// TIA Portal V18 export
DATA_BLOCK "FB10-Condition Check_1_DB"   // DB283
VERSION : 0.1
// stored: AutoNumber true, DBAccessibleFromOPCUA true, InstanceOfName FB10-Condition Check_1, InstanceOfType FB
"FB10-Condition Check_1"
   // VAR_INPUT
   //    "Time" : DInt;
   //    "Pump ON delay" : DInt;
   //    Check_Time { ExternalAccessible := 'False'; ExternalVisible := 'False'; ExternalWritable := 'False'} : DInt;
   //    Pressure_SP { ExternalAccessible := 'False'; ExternalVisible := 'False'; ExternalWritable := 'False'} : Real;
   //    Pressure_tolerance { ExternalAccessible := 'False'; ExternalVisible := 'False'; ExternalWritable := 'False'} : Real;
   //    Current_pressure { ExternalAccessible := 'False'; ExternalVisible := 'False'; ExternalWritable := 'False'} : Real;
   //    selected { ExternalAccessible := 'False'; ExternalVisible := 'False'; ExternalWritable := 'False'} : Bool;
   //    "Pressurising Tolerance" : Real;
   //    Pressurising_SP : Real;
   // END_VAR
   // VAR_OUTPUT
   //    "dispensing Time PV" : Int;
   //    "Checking Time pv" { ExternalAccessible := 'False'; ExternalVisible := 'False'; ExternalWritable := 'False'} : Int;
   //    Leaktest_ok { ExternalAccessible := 'False'; ExternalVisible := 'False'; ExternalWritable := 'False'} : Bool;
   //    Leaktest_nok { ExternalAccessible := 'False'; ExternalVisible := 'False'; ExternalWritable := 'False'} : Bool;
   //    Conditiontest_OK : Bool;
   //    Conditiontest_NOK { ExternalAccessible := 'False'; ExternalVisible := 'False'; ExternalWritable := 'False'} : Bool;
   //    "PAT @ installation" : DInt;
   //    Test_Data : "Condition_Check";
   // END_VAR
   // VAR_IN_OUT
   //    Commissioning_mode : Bool;
   //    "Start ConditonCheck" : Bool;
   //    "Stop ConditonCheck" : Bool;
   //    "ConditonCheck Running" : Bool;
   //    "ConditonCheck completed" : Bool;
   //    "ON Gear Pump" : Bool;
   //    "ON inlet" : Bool;
   //    Pressurising : Bool;
   //    run_rev : Bool;
   // END_VAR
   // VAR
   //    "dispensing time done" : Bool;
   //    "dispensing time in sec" : DInt;
   //    "timer input" : DInt;
   //    IEC_Timer_0_Instance_1 { S7_SetPoint := 'True'} : TON_TIME;
   //    IEC_Timer_0_Instance_2 { S7_SetPoint := 'True'} : TON_TIME;
   //    IEC_Timer_0_Instance_4 { S7_SetPoint := 'True'} : TON_TIME;
   //    "Press+ve" { ExternalAccessible := 'False'; ExternalVisible := 'False'; ExternalWritable := 'False'; S7_SetPoint := 'True'} : Real;
   //    "Press-ve" { ExternalAccessible := 'False'; ExternalVisible := 'False'; ExternalWritable := 'False'} : Real;
   //    IEC_Timer_0_Instance_3 { ExternalAccessible := 'False'; ExternalVisible := 'False'; ExternalWritable := 'False'; S7_SetPoint := 'True'} : TON_TIME;
   //    Checktime_ms { ExternalAccessible := 'False'; ExternalVisible := 'False'; ExternalWritable := 'False'; S7_SetPoint := 'True'} : DInt;
   //    Check_timesec { ExternalAccessible := 'False'; ExternalVisible := 'False'; ExternalWritable := 'False'} : DInt;
   //    temp_ons { ExternalAccessible := 'False'; ExternalVisible := 'False'; ExternalWritable := 'False'} : Bool;
   //    temp : Array[0..5] of Bool;
   //    IEC_Timer_0_Instance_5 { S7_SetPoint := 'True'} : TON_TIME;
   //    "WIth Tolerance" { S7_SetPoint := 'True'} : DInt;
   //    Pressure_achive_time : DInt;
   //    Pressure_ok : Bool;
   //    IEC_Timer_0_Instance { S7_SetPoint := 'True'} : TON_TIME;
   //    Result { S7_SetPoint := 'True'} : Bool;
   //    "result temp" : Bool;
   //    IEC_Timer_0_Instance_6 { S7_SetPoint := 'True'} : TON_TIME;
   //    Start_cond : Bool;
   //    IEC_Timer_0_Instance_7 { S7_SetPoint := 'True'} : TON_TIME;
   // END_VAR
BEGIN
END_DATA_BLOCK
